Fanuc KAREL source: ks00003.KL

-- PROVISIONAL review KL for V770-1; original PC SHA256 d2867b2447a35ee9ba52d7cfb76b996056e4204dd0e01b1fb750e91b8370e634
-- Incomplete behavior may be omitted. Consult companion uncertainty JSON. Do not deploy.
PROGRAM KS00003
%NOLOCKGROUP
VAR
  FLAG : BOOLEAN
  N : INTEGER
  STATUS : INTEGER
  PN : STRING[80]
  VN : STRING[80]
-- UNRESOLVED_DECL A type=001100
-- UNRESOLVED_DECL B type=001100
BEGIN
  -- UNRESOLVED_PC offsets 5-13; opcodes 3F,75
  -- UNRESOLVED_PC offsets 18-27; opcodes 3F,75
  -- UNRESOLVED_PC offsets 32-47; opcodes 22,22,30
  -- UNRESOLVED_PC offsets 52-56; opcodes 7F
END KS00003
